Omron CX-Programmer project NewProject (CX-Programmer 9.73)

# PLC NewPLC1: CP1L M

## Global symbols (name address type ; comment)
0.00 BOOL  ; START
0.01 BOOL  ; STOP
0.02 BOOL  ; SENSOR BATAS ATAS
0.03 BOOL  ; SENSOR BATAS BAWAH
0.04 BOOL  ; VALVE
0.06 BOOL  ; Proximity Conveyor
0.09 BOOL  ; Conveyor
100.00 BOOL  ; C1
100.01 BOOL  ; POMPA ON
100.02 BOOL  ; SENSOR BATAS ATAS
100.03 BOOL  ; SENSOR BATAS BAWAH
10.00 BOOL  ; C1
10.01 BOOL  ; BATAS ATAS
10.02 BOOL  ; BATAS BAWAH
W0.01 BOOL  ; Proximity Valve

## Program NewProgram1 (cyclic task 0)

### Section Section1

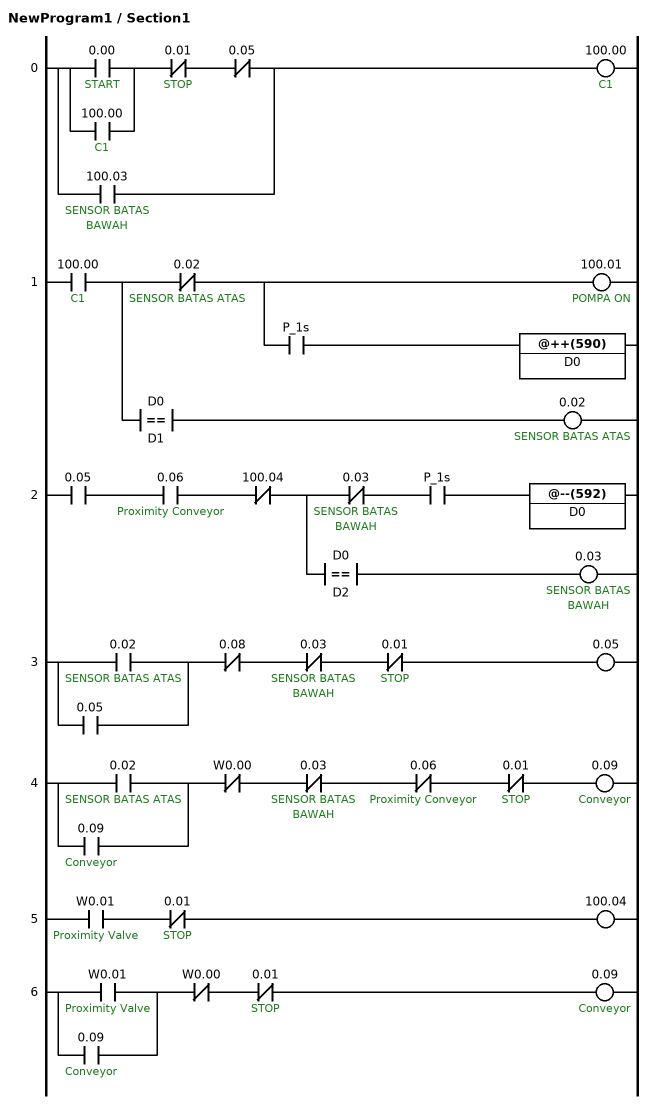
; rung 0
LD 0.00  ; START
OR 100.00  ; C1
ANDNOT 0.01  ; STOP
ANDNOT 0.05
OR 100.03  ; SENSOR BATAS BAWAH
OUT 100.00  ; C1
; rung 1
LD 100.00  ; C1
OUT TR0
ANDNOT 0.02  ; SENSOR BATAS ATAS
OUT 100.01  ; POMPA ON
AND P_1s
@++(590) D0
LD TR0
AND=(300) D0 D1
OUT 0.02  ; SENSOR BATAS ATAS
; rung 2
LD 0.05
AND 0.06  ; Proximity Conveyor
ANDNOT 100.04
OUT TR0
ANDNOT 0.03  ; SENSOR BATAS BAWAH
AND P_1s
@--(592) D0
LD TR0
AND=(300) D0 D2
OUT 0.03  ; SENSOR BATAS BAWAH
; rung 3
LD 0.02  ; SENSOR BATAS ATAS
OR 0.05
ANDNOT 0.08
ANDNOT 0.03  ; SENSOR BATAS BAWAH
ANDNOT 0.01  ; STOP
OUT 0.05
; rung 4
LD 0.02  ; SENSOR BATAS ATAS
OR 0.09  ; Conveyor
ANDNOT W0.00
ANDNOT 0.03  ; SENSOR BATAS BAWAH
ANDNOT 0.06  ; Proximity Conveyor
ANDNOT 0.01  ; STOP
OUT 0.09  ; Conveyor
; rung 5
LD W0.01  ; Proximity Valve
ANDNOT 0.01  ; STOP
OUT 100.04
; rung 6
LD W0.01  ; Proximity Valve
OR 0.09  ; Conveyor
ANDNOT W0.00
ANDNOT 0.01  ; STOP
OUT 0.09  ; Conveyor

### Section END
; rung 0
END(001)